// TIA Portal project "Mała" (V16)

(* hardware
DEVICE "S7-1200 station_1"  S7-1200 Station
   slot 0: "Rack_0"  S7-1200 Rack  Rack  V1.0
   slot 1: "PLC_1"  CPU 1214C DC/DC/DC  6ES7 214-1AG40-0XB0  V4.4
*)

// ===== PLC "PLC_1"  CPU 1214C DC/DC/DC =====

VAR_GLOBAL   // PLC tag table "Default tag table"
   "System_Byte" AT %MB1 : Byte;
   "FirstScan" AT %M1.0 : Bool;
   "DiagStatusUpdate" AT %M1.1 : Bool;
   "AlwaysTRUE" AT %M1.2 : Bool;
   "AlwaysFALSE" AT %M1.3 : Bool;
   "Clock_Byte" AT %MB0 : Byte;
   "Clock_10Hz" AT %M0.0 : Bool;
   "Clock_5Hz" AT %M0.1 : Bool;
   "Clock_2.5Hz" AT %M0.2 : Bool;
   "Clock_2Hz" AT %M0.3 : Bool;
   "Clock_1.25Hz" AT %M0.4 : Bool;
   "Clock_1Hz" AT %M0.5 : Bool;
   "Clock_0.625Hz" AT %M0.6 : Bool;
   "Clock_0.5Hz" AT %M0.7 : Bool;
   "Załączenie Zespołu Hydraulicznego I" AT %I0.0 : Bool;
   "Wyłączenie Zespołu Hydraulicznego" AT %I0.1 : Bool;
   "Sterowanie 2-Ręczne" AT %I0.2 : Bool;
   "Uszkodzenie Termiczne Zespołu Hydraulicznego" AT %I0.3 : Bool;
   "Spoczynkowa Pozycja Noża" AT %I0.4 : Bool;
   "Krańcowa Pozycja Noża" AT %I0.5 : Bool;
   "Położenie Spoczynkowe Siłownika Tasaka" AT %I0.6 : Bool;
   "Zatrzymanie Awaryjne/Otwarcie Pokrywy" AT %I0.7 : Bool;
   "Głowa w Maszynie" AT %I1.0 : Bool;
   "Zabezpiecznie Głowa Nie Za Duża" AT %I1.1 : Bool;
   "Załączenie Zespołu Hydraulicznego Q" AT %Q0.0 : Bool;
   "Główny Zawór Powietrza" AT %Q0.1 : Bool;
   "Siłownik Popychacza" AT %Q0.2 : Bool;
   "Siłownik Przemieszczenia Piły" AT %Q0.3 : Bool;
   "Siłownik Odcisku Noży" AT %Q0.4 : Bool;
   "Siłownik Tasaka" AT %Q0.5 : Bool;
   "Ogólna Awaria" AT %Q0.6 : Bool;
END_VAR

DATA_BLOCK "Zespół Cięcia Wstępnego_DB"   // DB1
{ S7_Optimized_Access := 'TRUE' }
VERSION : 0.1
// stored: InstanceOfName Zespół Cięcia Wstępnego
"Zespół Cięcia Wstępnego"
BEGIN
END_DATA_BLOCK

FUNCTION_BLOCK "Zespół Cięcia Wstępnego"   // FB1, SCL
{ S7_Optimized_Access := 'TRUE' }
VERSION : 0.1
   VAR_INPUT
      "Załączenie Zespołu Hydraulicznego I" : Bool;
      "Wyłączenie Zespołu Hydraulicznego" : Bool;
      "Sterowanie 2-Ręczne" : Bool;
      "Uszkodzenie Termiczne Zespołu Hydraulicznego" : Bool;
      "Spoczynkowa Pozycja Noża" : Bool;
      "Krańcowa Pozycja Noża" : Bool;
      "Położenie Spoczynkowe Siłownika Tasaka" : Bool;
      "Zatrzymanie Awaryjne/Otwarcie Pokrywy" : Bool;
      "Głowa w Maszynie" : Bool;
      "Zabezpiecznie Głowa Nie Za Duża" : Bool;
      "Brak Głowy / Za duża Głowa, Czas do Błędu" : Time := T#3s;
      "Opóźnienie Obrotu Noży" : Time := T#200ms;
      "Czas Docisku Tasaka" : Time := T#1s;
   END_VAR
   VAR_OUTPUT
      "Załączenie Zespołu Hydraulicznego Q" : Bool;
      "Główny Zawór Powietrza" : Bool;
      "Siłownik Popychacza" : Bool;
      "Siłownik Przemieszczenia Piły" : Bool;
      "Siłownik Odcisku Noży" : Bool;
      "Siłownik Tasaka" : Bool;
      "Ogólna Awaria" : Bool;
   END_VAR
   VAR
      Krok : Array[0..5] of Bool;
      "Numer Kroku" : Int;
      "old załączenie zespołu hydralicznego" : Bool;
      "zespół hydrauliczny" : Bool;
      "old sterowanie 2-ręczne" : Bool;
      "błąd głowy" : Bool;
      "błąd time" : TON_TIME;
      "obrót noży" : TON_TIME;
      "start obrotu noży" : TON_TIME;
      "docisk tasaka" : TON_TIME;
   END_VAR
   VAR_TEMP
      "t_załączenie zespołu hydraulicznego zbocze narastające" : Bool;
      "t_wyłączenie zespołu hydraulicznego" : Bool;
      "t_układ bezpieczny" : Bool;
      "t_sterowanie 2-ręczne zbocze narastające" : Bool;
      "t_start obrotu noży" : Bool;
      "t_koniec docisku tasaka" : Bool;
   END_VAR
   // Krok[0] := TRUE;
BEGIN
   REGION TRANZYCJE SPECJALNE
       REGION TS1 Załączenie Zespołu Hydraulicznego
           #"t_załączenie zespołu hydraulicznego zbocze narastające" :=
           #"Załączenie Zespołu Hydraulicznego I" AND
           NOT #"old załączenie zespołu hydralicznego";

           #"old załączenie zespołu hydralicznego" :=
           #"Załączenie Zespołu Hydraulicznego I";
       END_REGION

       REGION TS2 Wyłączenie Zespołu Hydraulicznego
           #"t_wyłączenie zespołu hydraulicznego" :=
           #"Zatrzymanie Awaryjne/Otwarcie Pokrywy" OR
           #"Wyłączenie Zespołu Hydraulicznego" OR
           "Uszkodzenie Termiczne Zespołu Hydraulicznego";

       END_REGION

       REGION TS3 Układ Bezpieczny
           #"t_układ bezpieczny" :=
           NOT #"Zatrzymanie Awaryjne/Otwarcie Pokrywy" AND
           #"zespół hydrauliczny" AND
           NOT "Uszkodzenie Termiczne Zespołu Hydraulicznego";

           //wyzwolony układ bezpieczeństwa, przerwij cykl
           IF NOT #"t_układ bezpieczny" THEN
               #"Numer Kroku" := 0;
           END_IF;
       END_REGION

       REGION T4 Sterowanie 2-ręczne Zbocze narastające 
           #"t_sterowanie 2-ręczne zbocze narastające" :=
           "Sterowanie 2-Ręczne" AND
           NOT #"old sterowanie 2-ręczne";

           #"old sterowanie 2-ręczne" := "Sterowanie 2-Ręczne";

       END_REGION

       REGION T5 Czas DO Błędu Za Dużej lub Braku Głowy           
           #"błąd time"(IN := #"Numer Kroku" = 2,
                        PT := #"Brak Głowy / Za duża Głowa, Czas do Błędu",
                        Q => #"błąd głowy");


       END_REGION
       REGION T6 Czas DO uruchomienia obrotu noży
           // Statement section REGION
           #"obrót noży"(IN := #"Numer Kroku" = 3 AND
                         NOT "Spoczynkowa Pozycja Noża" AND
                         #"Położenie Spoczynkowe Siłownika Tasaka",
                         PT := #"Opóźnienie Obrotu Noży",
                         Q => #"t_start obrotu noży");
       END_REGION

       REGION T7 
           // Statement section REGION
           #"docisk tasaka"(IN:=#"Numer Kroku" = 6,
                            PT:=#"Czas Docisku Tasaka",
                            Q=>#"t_koniec docisku tasaka");
       END_REGION

   END_REGION



   REGION GŁÓWNA SEKWENCJA
       CASE #"Numer Kroku" OF
           0: //Układ zabezpieczony
               //układ bezpieczeństwa nie jest wzbudzony,
               //nóż i tasak są w spoczynkowej pozycji
               IF #"t_układ bezpieczny" AND
                   "Spoczynkowa Pozycja Noża" AND
                   NOT #"Krańcowa Pozycja Noża" AND
                   #"Położenie Spoczynkowe Siłownika Tasaka" THEN
                   #"Numer Kroku" := 1;
               END_IF;
           1: //Stan gotowości do wystartowania

               //Nóż i Tasak w wyjściowej pozycji,
               //Klapa zamknięta i wciśnięty przycisk kolanowy,
               //oraz nie jest zadziałany czujnik popychacza
               IF "Spoczynkowa Pozycja Noża" AND
                   NOT #"Krańcowa Pozycja Noża" AND
                   #"Położenie Spoczynkowe Siłownika Tasaka" AND
                   #"t_sterowanie 2-ręczne zbocze narastające" AND
                   NOT "Zabezpiecznie Głowa Nie Za Duża" THEN
                   #"Numer Kroku" := 2;
               END_IF;

           2:  // Wyzwolony popychacz dociska głowę

               //Upłynął czas oczekiwnia na poprawną głowę, przerwij cykl
               IF #"błąd głowy" THEN
                   #"Numer Kroku" := 0;
               END_IF;

               //Czujnik popychacza i wykrycia głowy wyzwolone,
               //gdy nóż i tasak w pozycji startowej
               IF "Zabezpiecznie Głowa Nie Za Duża" AND
                   "Głowa w Maszynie" AND
                   "Spoczynkowa Pozycja Noża" AND
                   NOT #"Krańcowa Pozycja Noża" AND
                   #"Położenie Spoczynkowe Siłownika Tasaka" THEN
                   #"Numer Kroku" := 3;
               END_IF;
           3:  // Przemieszczanie noży

               //opóźniony obrót noży
               IF #"t_start obrotu noży" THEN
                   #"Numer Kroku" := 4;
               END_IF;
               ;
           4:  // Obrót noży + Przemieszczenie noży

               IF NOT "Spoczynkowa Pozycja Noża" AND
                   #"Krańcowa Pozycja Noża" THEN
                   #"Numer Kroku" := 5;
               END_IF;
               ;
           5:  // Powrót Noży
               IF "Spoczynkowa Pozycja Noża" AND
                   NOT #"Krańcowa Pozycja Noża" THEN
                   #"Numer Kroku" := 6;
               END_IF;
           6: //Docisk Tasaka

               //Przydełużony czas zadziałania Tasaka
               IF #"t_koniec docisku tasaka" THEN
                   #"Numer Kroku" := 0;
               END_IF;
       END_CASE;
   END_REGION

   REGION WYJŚCIA
       REGION Załączenie Zespołu Hydraulicznego
           IF #"t_wyłączenie zespołu hydraulicznego" THEN
               #"zespół hydrauliczny" := FALSE;
           ELSIF #"t_załączenie zespołu hydraulicznego zbocze narastające" THEN
               #"zespół hydrauliczny" := TRUE;
           END_IF;

           #"Załączenie Zespołu Hydraulicznego Q" :=
           #"zespół hydrauliczny";
       END_REGION

       REGION Główny Zawór Powietrza
           #"Główny Zawór Powietrza" :=
           True;
       END_REGION

       REGION Siłownik Popychacza
           #"Siłownik Popychacza" :=
           #"Numer Kroku" = 2 OR
           #"Numer Kroku" = 3 OR
           #"Numer Kroku" = 4 OR
           #"Numer Kroku" = 5 OR
           #"Numer Kroku" = 6;
       END_REGION

       REGION Siłownik Przemieszczenia Piły
           #"Siłownik Przemieszczenia Piły" :=
           #"Numer Kroku" = 3;
       END_REGION

       REGION Siłownik Odcisku Noży
           #"Siłownik Odcisku Noży" :=
           #"Numer Kroku" = 4;
       END_REGION

       REGION Siłownik Tasaka
           #"Siłownik Tasaka" :=
           #"Numer Kroku" = 6;
       END_REGION

       REGION Ogólna Awaria
           #"Ogólna Awaria" :=
           #"Uszkodzenie Termiczne Zespołu Hydraulicznego" OR
           #"Zatrzymanie Awaryjne/Otwarcie Pokrywy";
       END_REGION
   END_REGION
END_FUNCTION_BLOCK

ORGANIZATION_BLOCK "Main"   // OB1, LAD, ProgramCycle
TITLE = "Main Program Sweep (Cycle)"
{ S7_Optimized_Access := 'TRUE' }
VERSION : 0.1
   VAR_INPUT
      Initial_Call : Bool;   // Initial call of this OB
      Remanence : Bool;   // =True, if remanent data are available
   END_VAR
BEGIN

REGION Network 1 (SCL)
   "Zespół Cięcia Wstępnego_DB"("Załączenie Zespołu Hydraulicznego I":="Załączenie Zespołu Hydraulicznego I",
                                "Wyłączenie Zespołu Hydraulicznego":="Wyłączenie Zespołu Hydraulicznego",
                                "Sterowanie 2-Ręczne":="Sterowanie 2-Ręczne",
                                "Uszkodzenie Termiczne Zespołu Hydraulicznego":="Uszkodzenie Termiczne Zespołu Hydraulicznego",
                                "Spoczynkowa Pozycja Noża":="Spoczynkowa Pozycja Noża",
                                "Krańcowa Pozycja Noża":="Krańcowa Pozycja Noża",
                                "Położenie Spoczynkowe Siłownika Tasaka":="Położenie Spoczynkowe Siłownika Tasaka",
                                "Zatrzymanie Awaryjne/Otwarcie Pokrywy":="Zatrzymanie Awaryjne/Otwarcie Pokrywy",
                                "Głowa w Maszynie":="Głowa w Maszynie",
                                "Zabezpiecznie Głowa Nie Za Duża":="Zabezpiecznie Głowa Nie Za Duża",
                                "Załączenie Zespołu Hydraulicznego Q"=>"Załączenie Zespołu Hydraulicznego Q",
                                "Główny Zawór Powietrza"=>"Główny Zawór Powietrza",
                                "Siłownik Popychacza"=>"Siłownik Popychacza",
                                "Siłownik Przemieszczenia Piły"=>"Siłownik Przemieszczenia Piły",
                                "Siłownik Odcisku Noży"=>"Siłownik Odcisku Noży",
                                "Siłownik Tasaka"=>"Siłownik Tasaka",
                                "Ogólna Awaria"=>"Ogólna Awaria");
END_REGION
END_ORGANIZATION_BLOCK